{attribute 'GeneratedUsingTerminal: EL3022-0000-0016'}
{attribute addProperty BoxType "EL3022-0000-0016"}
{attribute addProperty Id "EtcSlaveTerminalBaseAI_Standard_Channel_1AT %I*AI_Standard_Channel_4A3944819AI_Standard_Channel_2AT %I*AI_Standard_Channel_4A3944819WcStateAT %I*WcState_9091E0EB2InfoDataAT %I*InfoData_32EB74EA10"}
{attribute addProperty CRC "1645147783"}
{attribute addProperty Size "30"}
TYPE EL3022_620EF687 EXTENDS EtcSlaveTerminalBase :
STRUCT
	{attribute addProperty Name "AI_Standard_Channel_1"}
	AI_Standard_Channel_1 : AI_Standard_Channel_4A394481;
	{attribute addProperty Name "AI_Standard_Channel_2"}
	AI_Standard_Channel_2 : AI_Standard_Channel_4A394481;
	{attribute addProperty Name "WcState"}
	WcState : WcState_9091E0EB;
	{attribute addProperty Name "InfoData"}
	InfoData : InfoData_32EB74EA;
END_STRUCT
END_TYPE

(* stored: Version 1.2.0.0, ProductVersion 3.1.4024.9
   DUT EL3022_620EF687: Id {18f7938c-81cc-41dd-83f3-a9f7e6ca63b6} *)
